FUNCTION_BLOCK T_GetComponentCompareResultsTrue EXTENDS T_UnitTestBase
VAR
  list : T_ComponentsCollection;
  newComponent : T_ComponentMock;
  actual : I_ComponentBase;
  expected : I_ComponentBase;
  result, tryGetResult : BOOL;
END_VAR

list.AddComponent(newComponent);

expected := newComponent;
tryGetResult := list.TryGetComponent(0, component => actual);

result := expected = actual;
assertion.AssertEquals_BOOL(TRUE, result, 'result := expected = actual');
assertion.AssertEquals_BOOL(TRUE, tryGetResult, 'tryGetResult');
TestFinished();

END_FUNCTION_BLOCK

(* stored: Version 1.1.0.1, ProductVersion 3.1.4024.12
   POU T_GetComponentCompareResultsTrue: Id {e9a4bf6b-918e-4c6c-8f6a-5af5f3d4eba8}, SpecialFunc None *)
